Universal Robots PolyScope program: APS2AndreGiBarros.urp

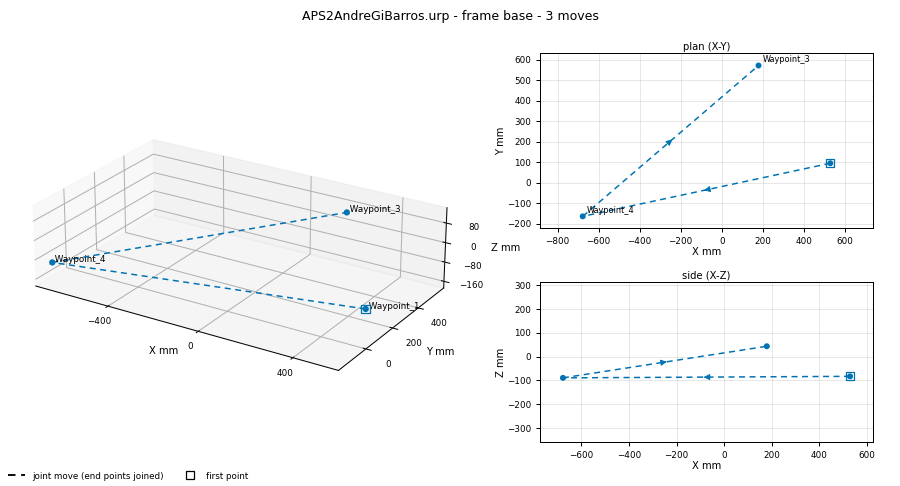
[picture p0: tool path of APS2AndreGiBarros.urp in frame base, 3 of 3 moves have a stored position in this frame; points joined in program order, loops and branches not executed]
Program APS2AndreGiBarros (installation=default directory=/programs/APS2OsUltimosRomanticos createdIn=3.15.3.106223 lastSavedIn=3.15.3.106223 robotSerialNumber=2017357017)
Calibrated DH parameters: a=[0.0001, -0.032836, -0.39033, 0.000086, 0.000053, 0]; d=[0.089393, 264.548863, -261.578988, -2.85966, 0.094927, 0.082356]; alpha=[1.569373, -0.001603, 0.013671, 1.570599, -1.570158, 0]; deltaTheta=[0.000031, -1.49356, 1.597104, -0.103695, -0.000023, -0.000043]
Robot Program (runOnlyOnce=false)
  produtos_caixa := 0
  var_loop := 0
  encaixotados := 0
  Loop Forever
    Loop While (checkContinuously=false) expression=var_loop<prod_na_cx
      Wait DigitalInput pin=digital_in[0]; digitalValue=1
      MoveJ speed 60 deg/s, acceleration 80 deg/s^2 (useActiveTCP=true)
        Waypoint Waypoint_1: TCP in base x=529.087 y=95.352 z=-82.529 mm, rx=0.0358 ry=-0.0362 rz=-0.0394 rad; joints [-182.82, -66.347, 116.608, -142.166, -87.479, 90.193] deg; flange x=522.738 y=89.036 z=97.248 mm, rx=0.0611 ry=3.1059 rz=0.0556 rad
        Call Pick
      produtos_caixa := produtos_caixa+1
      If produtos_caixa≥n_insp
        MoveJ speed 60 deg/s, acceleration 80 deg/s^2 (useActiveTCP=true)
          Waypoint Waypoint_4: TCP in base x=-677.611 y=-163.57 z=-88.987 mm, rx=-0.0509 ry=0.0554 rz=-3.0434 rad; joints [-354.836, -49.244, 86.983, -129.409, -91.627, 90.199] deg; flange x=-671.573 y=-169.833 z=90.802 mm, rx=-3.1011 ry=-0.1509 rz=0.0494 rad
        Set DigitalOutput pin=digital_out[2]; digitalValue=1
        Wait Sleep waitTime=0.5
        Set DigitalOutput pin=digital_out[2]; digitalValue=0
        Popup Message (haltProgram=false message=Fim da inspecao inputType=Text)
        produtos_caixa := 0
      Wait DigitalInput pin=digital_in[1]; digitalValue=1
      MoveJ speed 60 deg/s, acceleration 80 deg/s^2 (useActiveTCP=true)
        Waypoint Waypoint_3: TCP in base x=179.273 y=571.6 z=43.88 mm, rx=-0.0031 ry=-0.0121 rz=0.203 rad; joints [-117.847, -69.862, 97.399, -117.667, -89.947, 141.007] deg; flange x=177.339 y=571.987 z=223.869 mm, rx=-0.3173 ry=3.115 rz=-0.0051 rad
        Call Place
      var_loop := var_loop+1
      encaixotados := encaixotados+1
      Set ExpressionOutput pin=prod_encaixota; expression=encaixotados
    Set DigitalOutput pin=digital_out[1]; digitalValue=1
    Wait Sleep waitTime=0.5
    Set DigitalOutput pin=digital_out[1]; digitalValue=0
    var_loop := 0
SubProgram -> Place
SubProgram -> Pick
SubProgram Pick (keepSynchronizedWithDisk=false)
  Set DigitalOutput pin=tool_out[1]; digitalValue=0
  Set DigitalOutput pin=tool_out[0]; digitalValue=1
  Wait Sleep waitTime=0.5
SubProgram Place (keepSynchronizedWithDisk=false)
  Set DigitalOutput pin=tool_out[1]; digitalValue=1
  Set DigitalOutput pin=tool_out[0]; digitalValue=0
  Wait Sleep waitTime=0.5
